ABB RobotStudio station: Solution final version.rsstn

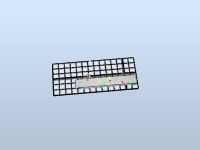
Station Solution4 (saved by RobotStudio 6.8.8148.134)
Controller System1, task T_ROB1: task frame (RAPID world) sits at (5535.63, 749.82, 709.58) mm in the station
Controller System1
  mechanical unit ROB_1: IRB1600_10_145__01, 6 joints, base frame (480.91, -394.38, -359.58) mm, rotated rx 0 ry 0 rz 90 deg
  mechanical unit CNV1: ?, 1 joints, base frame (0, 0, 0) mm
Layout (positions relative to the parent item):
  - bin mover_3 [smart component] at (-500, 0, 0) mm
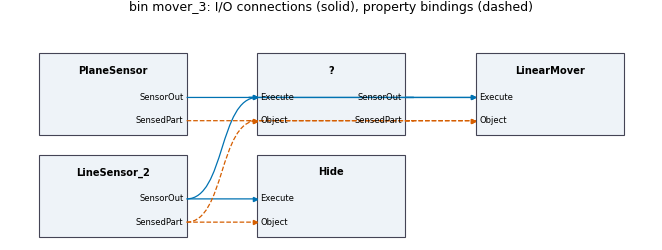
      connections:
        ?.SensorOut -> LinearMover.Execute
        PlaneSensor.SensorOut -> LinearMover.Execute
        ?.SensorOut -> ?.Execute
        LineSensor_2.SensorOut -> ?.Execute
        LineSensor_2.SensorOut -> Hide.Execute
        ?.SensedPart => LinearMover.Object
        PlaneSensor.SensedPart => LinearMover.Object
        ?.SensedPart => ?.Object
        LineSensor_2.SensedPart => ?.Object
        LineSensor_2.SensedPart => Hide.Object
    - LinearMover [smart component, from Components\LinearMover.rslib] at (6663.26, 677.27, 1050.93) mm, rotated rx 180 ry 0 rz 90 deg
        properties: Object=(none); Direction=[0 0 -1]; Speed=8; Reference=Global; ReferenceObject=(none)
    - PlaneSensor [smart component, from Components\PlaneSensor.rslib]
        properties: Origin=[7.419145 0.146999 1.42]; Axis1=[0 0 -1.35]; Axis2=[0 0.4 0]; SensedPart=(none)
      - _sensorPart_ [part]
    - LineSensor_2 [smart component, from Components\LineSensor.rslib]
        properties: Start=[7.369145 0.346999 0.008]; End=[7.369145 0.346999 0.123]; Radius=0.09; SensedPart=(none); SensedPoint=[0 0 0]
      - _sensorPart_ [part]
    - Hide [smart component, from Components\Hide.rslib]
        properties: Object=(none)
  - bin1_2 [part] at (6733.74, 347, -12) mm
  - conveyor 1 [part] at (-3500, -1500, -4460) mm, rotated rx 90 ry 0 rz 90 deg
  - Suction gripper 18cm [smart component] at (6727.84, 418.35, 1386.5) mm, rotated rx 180 ry 0 rz -90 deg
      signals: DI do1
      connections:
        Suction gripper 18cm.do1 -> LogicGate.InputA
        Suction gripper 18cm.do1 -> LineSensor.Active
        LogicGate.Output -> Detacher.Execute
        LineSensor.SensorOut -> Attacher.Execute
        Attacher.Executed -> ?.Set
        Detacher.Executed -> ?.Reset
        LineSensor.SensedPart => Attacher.Child
        Attacher.Child => Detacher.Child
    - Attacher [smart component, from Components\Attacher.rslib]
        properties: Parent=Suction_gripper 18cm; Flange=0; Child=Yellow block; Mount=false; Offset=[0 0 0]; Orientation=[0 0 0]
    - LogicGate [smart component, from Components\LogicGate.rslib]
        properties: Operator=NOT; Delay=0
    - LineSensor [smart component, from Components\LineSensor.rslib] at (7150.29, 306.47, 1168.39) mm, rotated rx 180 ry 0 rz 90 deg
        properties: Start=[-0.30577796087058 -7.14894421240012 1.16938863540814]; End=[-0.305777964813962 -7.14894420825673 1.13938863540814]; Radius=0.09; SensedPart=Yellow block; SensedPoint=[6.48149609375 0.691603332519531 1.22920129394531]
      - _sensorPart_ [part]
    - Detacher [smart component, from Components\Detacher.rslib]
        properties: Child=Yellow block; KeepPosition=true
  - Suction_gripper 18cm [mechanism] at (6727.84, 418.35, 1471.5) mm, rotated rx 180 ry 0 rz -90 deg
      TCP Suction_gripper_18cm at (90, 0, 90) mm, rotated rx 90 ry 0 rz 0 deg
      links: Suction gripper 18cm
  - IRB1600_10_145__01 [mechanism] at (6016.55, 355.44, 350) mm, rotated rx 0 ry 0 rz 90 deg; joint values [-1.4826, -0.0513, 0.0498, 0, 1.5723, -1.4826] (rad or m)
      links: Base, Link1, Link2, Link3, Link4, Link5, Link6
  - Position tracker [smart component]
      signals: DI do_rapid
      connections:
        LineSensor.SensorOut -> RapidVariable.Set
        PlaneSensor_3.SensedPart => LinearMover.Object
        PlaneSensor_3.SensedPart => PositionSensor_2.Object
        LineSensor.SensedPart => PositionSensor_2.Object
        PositionSensor_2.Position => VectorConverter.Vector
        VectorConverter.Y => RapidVariable.Value
    - RapidVariable [smart component, from Components\RapidVariable.rslib]
        properties: DataType=num; Controller=System1; Task=T_ROB1; Module=Module1; Variable=y; Value=0.454144435518621
    - PositionSensor_2 [smart component, from Components\PositionSensor.rslib]
        properties: Object=(none); Reference=Object; ReferenceObject=Reference; Position=[-0.775833999989715 0.454144435518621 -0.741395]; Orientation=[0 0 0]
    - LineSensor [smart component, from Components\LineSensor.rslib]
        properties: Start=[5.101063 2.339147 0.72958]; End=[5.101063 0.739147 0.72958]; Radius=0.02; SensedPart=(none); SensedPoint=[0 0 0]
      - _sensorPart_ [part]
    - VectorConverter [smart component, from Components\VectorConverter.rslib]
        properties: X=-0.775833999989715; Y=0.454144435518621; Z=-0.741395; Vector=[-0.775833999989715 0.454144435518621 -0.741395]
  - Reference [part] at (3022.67, -346.33, 752.97) mm
  - Random position [smart component]
      connections:
        PlaneSensor.SensorOut -> Random.Execute
        PlaneSensor.SensorOut -> LinearMover.Execute
        PlaneSensor.SensedPart => LinearMover.Object
        Random.Value => LinearMover.Speed
    - Random [smart component, from Components\Random.rslib]
        properties: Value=-0.154648786715534; Min=-0.3; Max=1.05
    - PlaneSensor [smart component, from Components\PlaneSensor.rslib] at (-2700, 0, 0) mm
        properties: Origin=[4.525795 0.752121 0.710084]; Axis1=[0 0 0.18]; Axis2=[0 1.575 0]; SensedPart=(none)
      - _sensorPart_ [part]
    - LinearMover [smart component, from Components\LinearMover.rslib]
        properties: Object=(none); Direction=[0 0.001 0]; Speed=-0.154648786715534; Reference=Global; ReferenceObject=(none)
  - 输送链_2 [conveyor]
    - Yellow block [part] at (0, -475.41, 0) mm
    - 传送带对象_20 [conveyorobject] at (7814.83, 749.82, 709.58) mm
      - Yellow block [part] at (634.96, -1786.69, -1311.3) mm
    - 传送带对象_21 [conveyorobject] at (6114.83, 749.82, 709.58) mm
      - Yellow block [part] at (910.79, -1788.36, -1308.19) mm
    - 传送带对象_22 [conveyorobject] at (4414.83, 749.82, 709.58) mm
      - Yellow block [part] at (898.39, -1645.14, -1310.57) mm
    - 传送带对象_23 [conveyorobject] at (2714.83, 749.82, 709.58) mm
      - Yellow block [part] at (976.48, -1766.47, -153.96) mm
    - 传送带对象_24 [conveyorobject] at (1014.83, 749.82, 709.58) mm
      - Yellow block [part] at (300, -614.69, -698) mm
    - 传送带对象_25 [conveyorobject] at (-685.17, 749.82, 709.58) mm
      - Yellow block [part] at (300, -1197.79, -698) mm
  - conveyor base [smart component]
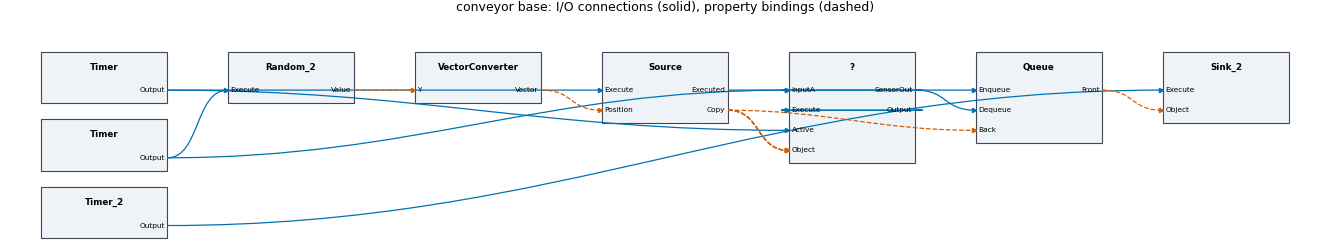
      connections:
        Timer.Output -> Source.Execute
        Source.Executed -> Queue.Enqueue
        ?.SensorOut -> ?.InputA
        ?.Output -> ?.Execute
        ?.SensorOut -> Queue.Dequeue
        ?.Output -> ?.Execute
        Timer.Output -> ?.InputA
        Timer.Output -> ?.Active
        Timer.Output -> Random_2.Execute
        Timer_2.Output -> Sink_2.Execute
        Source.Copy => ?.Object
        Source.Copy => ?.Object
        Source.Copy => ?.Object
        Source.Copy => ?.Object
        Source.Copy => Queue.Back
        Random_2.Value => VectorConverter.Y
        VectorConverter.Vector => Source.Position
        Queue.Front => Sink_2.Object
    - Queue [smart component, from Components\Queue.rslib]
        properties: Back=box random 1_62; Front=(none); Queue={e48e581f-8a66-4fec-b269-07e351db24a9};{4c3ea5d8-6def-4fc0-8f82-46bd2df239bd};{ba08add5-bbba-4563-8d87-2a4216425c02};{1608ad6a-3bb8-4e45-842f-0db6d97c7998};{f677491c-453d-4a4f-af0a-64563ff1f7ae};{bc5b26f6-3573-408f-a660-dd5e97df8b32};{84b58e33-0abf-440c-990d-e526580a760c};{d3b7469e-b0dc-40b0-a06e-beae69c32c93};{30de592b-dd57-4fe6-8609-591667023966};{67c6b656-de77-4921-91bd-a3a583d0da80};{488b8de9-8c86-42ee-972b-08a20bd55542};{18e44fb0-5c04-4911-8fdb-56f335ea8d72};{77774b90-ba08-47c6-8ad1-885a7e1fb4a1};{6a948890-dbed-4162-bb6d-d1a3b98f93da};{725da25f-aeb6-49d9-ad59-fd2d27d00660};{c0ccced7-8566-4310-97fe-e94f1994ccc8};{b944b4ba-03b2-4a3e-afd4-f216425226b1};{27b7961a-324a-4e87-b51b-237e4153a626};{702a0380-ebb8-45f7-b564-6161fbe14c88};{b06d3921-15de-44ac-82dd-5aa6a0e8191c};{b62c3fb7-8e55-4cdf-9d67-d4cc2f5ef05a};{92b684de-77f5-47ec-9555-be1b7a48fbe3};{7dd309d7-c641-401f-8e8f-2943d99e045b};{f6cbf723-84a9-4360-92db-7eacec9b81eb};{8f04e364-2d0b-4387-a572-90ab264d713a};{f2b8ee8f-9390-4fe2-b2ab-eaf01b7b0b47};{d9b300c1-4931-4bda-93de-414dafeee843};{6206577c-5e6c-43f3-88f3-e1b3bd454b62};{ba872c81-b989-472b-a4ac-fc6784b3217f};{56451b1c-727d-446b-9b60-68fa0f3418b4};{2296976c-1bbb-42f7-aeb4-7a1bba6c9a4a};{c66dc883-a25e-4f76-9ff4-008f9fa005f6};{aa2e9503-91f7-4371-a350-06b37842132b};{7e4f5268-017a-4f3c-9efe-60754f5d1d82};{e2a3c9ab-37c7-43a7-a13a-7397987f7ad5};{f528e014-3432-4e8f-8fe3-02ce617fcae9};{26e30cde-814d-40ae-b1a8-5c66cde7944b};{0b00fac2-6d35-4e26-9e24-a885e653ff60};{2542b8e2-fb6f-4b5a-b318-5a4e39e838ff};{99c9a211-fffe-44bf-9231-65058f9b545b};{73949de5-1df1-47bb-94da-e36fd1d8012d};{367b4e6f-f14c-457e-9fff-9ba529f51609};{a7cfef54-575f-4f30-a9a2-3ca4443502d7};{83fe5157-9726-4242-982a-904829c1a194};{bed63ce3-0f35-400f-9e5f-341d4225a442};{f437f502-005c-4b18-8595-7a5e4b2f9866};{b105fff9-5524-4476-ba9a-dfc6d9239c7c};{42045499-c356-43b6-838a-509ee5b1abe9};{31ccd5bb-9d2f-4ed1-9e19-94ce33b3bac9};{2960c81f-3f27-4772-8f80-2c98e67730ff};{7be1523c-6d8e-4136-bb31-f51b211182fb};{d7610290-98d3-4acb-8121-9071e0bc94d1};{3a5b0821-40b0-4715-a1ad-5a183596995f};{8c755288-18e4-4f97-8f2e-27b2742b70fa};{ee6e5577-30f4-4adc-85ac-cf38aea0e1e6};{f78435b0-db07-4bbc-b5bc-85e03782103c};{90f284d8-8738-4acd-be7f-98b56e1f0d3f};{9d98be80-3ca0-48d7-9d3c-cefffa3d1c93};{f822d83b-f9df-4b16-b601-fa0d0dffa441};{bb19192c-fa2f-4981-8aa1-10d2868712e5};{1cf355de-6181-4349-92a7-6e94814f8d48};{bae2d34c-ccd3-4cf7-a2cb-48542c7e17bd};{8541b48a-3765-4fcd-80c7-82fec0d416b5};{0be9d16c-7211-4316-a459-bb1d6514ca7b};{e7c7b897-b10b-4d0b-a94e-cde444c8761f};{6606d5da-442b-48b0-82dd-9b9b8062e5de};{6ef14163-b9e0-446f-8dfb-c6bf757800c4};{b1e4ca14-3f36-4439-b0af-a86262123063};{1d96b994-e8db-43b5-bce2-7ee11b647908};{0658f03b-5339-4ba3-bba5-da09f969777a};{391cacbe-1cc6-4825-bec9-4b5f2e5b84b0};{0744154e-d6d3-4638-ab4f-c693baed92d0};{0843ab46-09f0-40bf-b006-27e756fddc51};{9b4d8454-b44a-4c8a-a6b3-9fe29a173b69};{a11b88d0-dd92-462c-83d6-978b9f3471ae};{6ccc8720-4f16-4012-80bb-fcf442773d5f};{e210b5ec-84ed-4b94-9572-b22f3fbcc127};{39acf8ba-ac97-411b-88c8-0169cc681850};{6d5ff900-1c8b-40a1-aac4-52a4b0636b62};{82d10434-83ba-4ccd-a81f-f55b320888d2};{8c7fc2bc-dc19-4362-96a0-73f77254a46a};{cf8bff45-354d-4ef6-a704-58d35056d60a};{cff74c0b-f486-4f81-9669-93d729b8a6ac};{a6959f27-b5af-470d-be35-478272a360fd};{e9b7b5cf-058a-4499-8115-f51533c1ce43};{ea88c957-555c-4901-a709-50ca76df20aa};{bb874c55-ddb4-4dca-a01c-f28617aadc21};{f7d15137-90d4-4e34-9aff-829f4d21f2b3};{08986ffa-bc34-48d2-a759-06500ca70ddc};{bbe67ba7-d6b4-48cc-8374-75a94dafd8e2};{7d866e28-ba7c-4dcf-a01f-8cf9da0ffbd7};{c2d493b3-fec8-41ae-ad8a-96fb1031a3a8};{44aee37b-b427-49cb-86b0-52d50a98a895};{c8bd1ada-3109-4d88-8660-aefe2cdb22b4};{f2357b95-57c3-4d8a-a240-e25c246e0195};{e76cdebb-4b15-4c1c-84c0-8fe687a52d2a};{cacb030a-d6b9-4f14-a219-c2944cd19772};{3e97ad68-ab79-4a3a-bb78-e0e4b81befe7};{a960feb5-2d0c-4805-9613-0331805c739b};{60fce2f8-46ed-456a-aa54-76d6421e5c87};{1c294a21-0b9e-4b7f-9207-770e040456a7};{38a7fee2-987e-4c1a-a0b8-1a7b4ae1ce5d};{9e064271-f182-43f4-a0b0-83f4f1ad4b7a};{42ae712b-f6e4-459b-9a97-9faff141fcbb}; NumberOfObjects=5
    - Source [smart component, from Components\Source.rslib] at (0, 5000, 0) mm
        properties: Source=box random 1; Copy=box random 1_62; Parent=(none); Position=[0 -0.0803998819693923 0]; Orientation=[0 0 0]; Transient=false; PhysicsBehavior=0
    - Timer [smart component, from Components\Timer.rslib]
        properties: StartTime=0; Interval=2; Repeat=true; CurrentTime=5.16
    - LinearMover [smart component, from Components\LinearMover.rslib]
        properties: Object=Queue; Direction=[0.1 0 0]; Speed=1; Reference=Global; ReferenceObject=(none)
    - Timer [smart component, from Components\Timer.rslib]
        properties: StartTime=0.1; Interval=2; Repeat=true; CurrentTime=5.16
    - Random_2 [smart component, from Components\Random.rslib]
        properties: Value=-0.0803998819693923; Min=-0.75; Max=0.75
    - VectorConverter [smart component, from Components\VectorConverter.rslib]
        properties: X=0; Y=-0.0803998819693923; Z=0; Vector=[0 -0.0803998819693923 0]
    - Timer_2 [smart component, from Components\Timer.rslib]
        properties: StartTime=0; Interval=2; Repeat=true; CurrentTime=5.16
    - Sink_2 [smart component, from Components\Sink.rslib]
        properties: Object=(none)
  - conveyor base_2 [smart component]
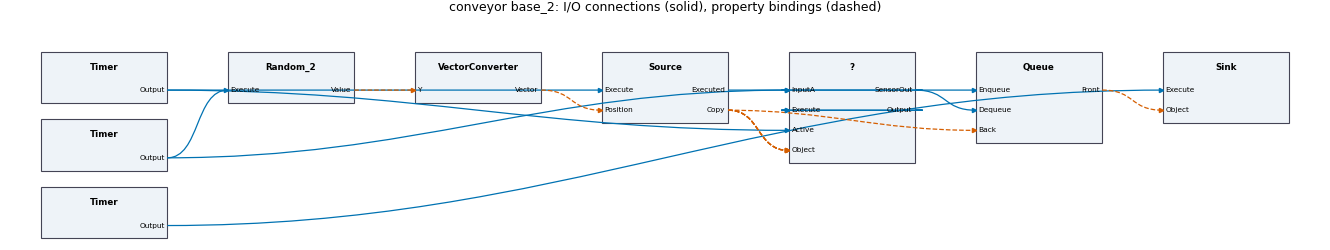
      connections:
        Timer.Output -> Source.Execute
        Source.Executed -> Queue.Enqueue
        ?.SensorOut -> ?.InputA
        ?.Output -> ?.Execute
        ?.SensorOut -> Queue.Dequeue
        ?.Output -> ?.Execute
        Timer.Output -> ?.InputA
        Timer.Output -> ?.Active
        Timer.Output -> Random_2.Execute
        Timer.Output -> Sink.Execute
        Source.Copy => ?.Object
        Source.Copy => ?.Object
        Source.Copy => ?.Object
        Source.Copy => ?.Object
        Source.Copy => Queue.Back
        Random_2.Value => VectorConverter.Y
        VectorConverter.Vector => Source.Position
        Queue.Front => Sink.Object
    - Queue [smart component, from Components\Queue.rslib]
        properties: Back=box random 2_63; Front=(none); Queue={e48e581f-8a66-4fec-b269-07e351db24a9};{4c3ea5d8-6def-4fc0-8f82-46bd2df239bd};{ba08add5-bbba-4563-8d87-2a4216425c02};{1608ad6a-3bb8-4e45-842f-0db6d97c7998};{f677491c-453d-4a4f-af0a-64563ff1f7ae};{bc5b26f6-3573-408f-a660-dd5e97df8b32};{84b58e33-0abf-440c-990d-e526580a760c};{d3b7469e-b0dc-40b0-a06e-beae69c32c93};{30de592b-dd57-4fe6-8609-591667023966};{67c6b656-de77-4921-91bd-a3a583d0da80};{488b8de9-8c86-42ee-972b-08a20bd55542};{18e44fb0-5c04-4911-8fdb-56f335ea8d72};{77774b90-ba08-47c6-8ad1-885a7e1fb4a1};{6a948890-dbed-4162-bb6d-d1a3b98f93da};{725da25f-aeb6-49d9-ad59-fd2d27d00660};{c0ccced7-8566-4310-97fe-e94f1994ccc8};{b944b4ba-03b2-4a3e-afd4-f216425226b1};{27b7961a-324a-4e87-b51b-237e4153a626};{702a0380-ebb8-45f7-b564-6161fbe14c88};{b06d3921-15de-44ac-82dd-5aa6a0e8191c};{b62c3fb7-8e55-4cdf-9d67-d4cc2f5ef05a};{92b684de-77f5-47ec-9555-be1b7a48fbe3};{7dd309d7-c641-401f-8e8f-2943d99e045b};{f6cbf723-84a9-4360-92db-7eacec9b81eb};{8f04e364-2d0b-4387-a572-90ab264d713a};{f2b8ee8f-9390-4fe2-b2ab-eaf01b7b0b47};{d9b300c1-4931-4bda-93de-414dafeee843};{6206577c-5e6c-43f3-88f3-e1b3bd454b62};{ba872c81-b989-472b-a4ac-fc6784b3217f};{56451b1c-727d-446b-9b60-68fa0f3418b4};{2296976c-1bbb-42f7-aeb4-7a1bba6c9a4a};{c66dc883-a25e-4f76-9ff4-008f9fa005f6};{aa2e9503-91f7-4371-a350-06b37842132b};{7e4f5268-017a-4f3c-9efe-60754f5d1d82};{e2a3c9ab-37c7-43a7-a13a-7397987f7ad5};{f528e014-3432-4e8f-8fe3-02ce617fcae9};{26e30cde-814d-40ae-b1a8-5c66cde7944b};{0b00fac2-6d35-4e26-9e24-a885e653ff60};{2542b8e2-fb6f-4b5a-b318-5a4e39e838ff};{99c9a211-fffe-44bf-9231-65058f9b545b};{73949de5-1df1-47bb-94da-e36fd1d8012d};{367b4e6f-f14c-457e-9fff-9ba529f51609};{a7cfef54-575f-4f30-a9a2-3ca4443502d7};{83fe5157-9726-4242-982a-904829c1a194};{bed63ce3-0f35-400f-9e5f-341d4225a442};{f437f502-005c-4b18-8595-7a5e4b2f9866};{9a0cab65-2397-4188-bc41-cf652fbf8898};{941c0970-3b80-4489-9148-16d5d3c95db8};{5ba0f877-d6ea-493b-a2f1-443817ea1bdf};{5de72a40-24d3-4735-a83e-140ebadfa059};{fa8c35bd-2a9a-44f8-9b58-73b3deb4511a};{95fc4834-c60d-41e2-95b1-62a856343879};{4a4b129d-b181-4d11-9bce-364b45794abd};{1d13c647-9247-481a-9323-002b2efab1f2};{5d5ac231-d74a-481f-9d60-d4ed3c609295};{9c232dc5-cafb-49dc-ac7d-49f9565aa061};{0a610a08-cf6b-4e99-973b-5bba28012cfb};{9aa8b73c-1d04-4bc2-86d7-2d31a4418e36};{d67df86c-620e-48fb-b812-fb4ad1e7dea9};{65483b71-b5f9-4883-ad12-420147a524aa};{85d671a5-ba29-4c0e-87e1-d9b33fa823f9};{92a71b09-30ab-475c-8933-9e5f01295ec4};{a00b1944-3818-45cc-9475-2d09b52e653b};{b145dda1-fbf5-4e62-a73c-395e30d6dd69};{6dddc38c-222b-40f2-91b0-876980f40815};{2b9da836-4bf5-4d8f-ac74-2d28f0eb4e51};{517ac4c7-4730-4cb0-a707-f87587d789f2};{0f0d7c83-f1ce-48fb-a80b-b22b544eee9b};{f9e0bd1a-328c-43db-b665-713982ad9551};{4c6e7a35-81c2-4c02-8628-6e8b68811b28};{723f4bec-1bc4-46b9-80c9-94c7c97e6454};{e5d5d3a1-be73-488a-a9ff-8ffeaf9cc457};{2521d265-1639-483e-8429-4f96a8802b6f};{3a375944-9a19-4e04-ba94-a4697befbc04};{dfa99347-922b-4406-916c-a23705f6f694};{f41de96e-135c-4ff1-a0f1-ac25ca0b4fbd};{61d4a249-e0a5-49d4-926a-58f802f4d981};{2070fa79-0f33-4b67-9598-bd35bf8d01ed};{43a1226d-b2a1-4972-856b-657db23b8e0a};{30775785-8cc2-4888-a456-e2853ec74311};{77809f03-2db0-4855-a9cd-199abe1bf4a6};{82b6306a-5718-4a32-8421-873217a824ce};{c284f025-2489-4344-a964-97ebee5d4451};{034aea7d-e78e-459c-9640-913c75fdb37e};{358ee115-9f46-41b7-ba1a-a96a4d507549};{c789a6de-4596-450d-926d-4b96ca7da022};{b275474e-bb4c-40a5-9de3-f3cacea9b337};{9e5b3e5d-3bb7-4c53-b001-a44e97753210};{5938a1ac-9741-4ae6-a44a-cfbeddd30ab1};{844fd4f9-ad00-4033-ba36-df8f5de7e3a4};{288418bc-a86d-4b16-a5fb-478b2ea2d971};{1bfa687d-06df-4a77-92d3-2683f829d4e3};{80d3484b-a7c2-45f9-af67-0e34bcfd6f68};{69052e92-6335-4a1a-921d-a9a3ca289a2f};{6d8bf7b5-6c08-4b3f-b1c8-7f931c8617a8};{56fa55c3-7825-42e7-8904-b93f621254d8};{99116da4-144c-47f1-a42d-1d777de07b72};{e27173cc-98be-4083-ad1e-b896e7511c30};{77931f39-9253-4c97-8851-97293684fc48};{1578d08e-c182-4eae-a940-784364c44454};{3d0d464e-2357-498a-a26a-a575e9d84ee5};{d9fb72da-3f5e-4077-9ec9-18dfd300d7a7};{f26423e1-4853-42af-b915-30a42f579b9c};{6ef03125-0d10-4204-adca-0569244197c0};{eb959d8b-76fe-413c-8a45-043fcaadba30};{cd79a4e2-bf91-4b03-b1c3-ea94a0243daa};{32063103-f801-44f5-b808-3248e0d4b6da};{aeba722b-5807-49cd-96b6-9ffc5e4578ec};{d1d9545e-8b4f-4c85-bdf5-413f7d2a04b0};{22d2ded6-1d2c-407e-bba2-a44af4b299f1};{6acc5802-14b2-4e38-acf3-01ca714794b4}; NumberOfObjects=5
    - Source [smart component, from Components\Source.rslib] at (0, 5000, 0) mm
        properties: Source=box random 2; Copy=box random 2_63; Parent=(none); Position=[0 0.170611426662938 0]; Orientation=[0 0 0]; Transient=false; PhysicsBehavior=0
    - Timer [smart component, from Components\Timer.rslib]
        properties: StartTime=1; Interval=2; Repeat=true; CurrentTime=5.16
    - LinearMover [smart component, from Components\LinearMover.rslib]
        properties: Object=Queue; Direction=[0.1 0 0]; Speed=1; Reference=Global; ReferenceObject=(none)
    - Timer [smart component, from Components\Timer.rslib]
        properties: StartTime=1.1; Interval=2; Repeat=true; CurrentTime=5.16
    - Random_2 [smart component, from Components\Random.rslib]
        properties: Value=0.170611426662938; Min=-0.75; Max=0.75
    - VectorConverter [smart component, from Components\VectorConverter.rslib]
        properties: X=0; Y=0.170611426662938; Z=0; Vector=[0 0.170611426662938 0]
    - Timer [smart component, from Components\Timer.rslib]
        properties: StartTime=1; Interval=2; Repeat=true; CurrentTime=5.16
    - Sink [smart component, from Components\Sink.rslib]
        properties: Object=(none)
  - box random 1 [part]
  - box random 2 [part]
  - box random 2_57 [part] at (7888, -139.09, 0) mm
  - box random 1_58 [part] at (6888, -484.74, 0) mm
  - box random 2_59 [part] at (4160, 269.69, 0) mm
  - box random 1_60 [part] at (3160, 19.41, 0) mm
  - box random 2_61 [part] at (2160, -32.02, 0) mm
  - box random 1_62 [part] at (1160, 425.58, 0) mm
  - box random 2_63 [part] at (160, 592.8, 0) mm
Attachment: Suction gripper 18cm is attached to Suction_gripper 18cm / Suction gripper 18cm
Attachment: Suction_gripper 18cm is attached to IRB1600_10_145__01 / Link6
Attachment: Yellow block is attached to Suction_gripper 18cm / Suction gripper 18cm
Conveyor tracking 连接_2: unit CNV1, TravelOffset=7.2, QueueTrackDistance=0, StartWindowWidth=1.8, SyncSeparation=0, CountsPerMeter=10000
Station logic (signal -> signal, property => property):
  System1.do_attach -> Suction gripper 18cm.do1
Targets, tools, work objects and paths stored in the station, written as RAPID:
! task T_ROB1
MODULE Module1
  PERS tooldata Suction_gripper_18cm:=[TRUE,[[0,0,85],[1,0,0,0]],[1,[0,0,1],[1,0,0,0],0,0,0]];
  CONST robtarget Target_10:=[[480.915,355.615,676.92],[0,-0.707106781,0.707106781,0],[0,0,0,0],[9E+09,9E+09,9E+09,9E+09,9E+09,0]];
  CONST robtarget Target_20:=[[-70.300373856,355.874016057,111.580012181],[-0.000000002,0.707106781,-0.707106781,0.000000007],[0,-1,0,0],[9E+09,9E+09,9E+09,9E+09,9E+09,0]];
  CONST robtarget Target_30:=[[1192.207950487,-331.467717415,676.919992598],[0.000000021,0.707106781,-0.707106781,0.000000022],[-1,-1,-1,0],[9E+09,9E+09,9E+09,9E+09,9E+09,0]];
  PROC Path_10()
    MoveL Target_10,vmax,fine,Suction_gripper_18cm\WObj:=wobj0;
    MoveL reltool(Target_20,-y*1000,0,0),vmax,z10,Suction_gripper_18cm\WObj:=wobj_cnv1;
    Set do_attach;
    MoveL Target_30,vmax,fine,Suction_gripper_18cm\WObj:=wobj0;
    Reset do_attach;
    MoveL Target_10,vmax,fine,Suction_gripper_18cm\WObj:=wobj0;
  ENDPROC
  PROC main()
    ActUnit CNV1;
    WaitWObj wobj_cnv1;
    Path_10;
    DropWObj wobj_cnv1;
  ENDPROC
ENDMODULE

! task T_ROB1
MODULE CalibData
  TASK PERS wobjdata wobj_cnv1:=[FALSE,FALSE,"CNV1",[[0,0,0],[1,0,0,0]],[[0,0,0],[1,0,0,0]]];
ENDMODULE

